TYPE ST_AxisHaltParameter EXTENDS ST_AxisStopParameter :
STRUCT
	eBufferMode: MC_BufferMode := MC_Aborting;
END_STRUCT
END_TYPE

(* stored: Version 1.1.0.1, ProductVersion 3.1.4020.12
   DUT ST_AxisHaltParameter: Id {6c7bcecd-3bfd-432d-b499-a45d72c40d87} *)
